// TIA Portal V18 export
VAR_GLOBAL   // PLC tag table "Default tag table"
   "Alarm Drive1" AT %I0.0 : Bool;
   "Alarm Drive 2" AT %I0.1 : Bool;
   setFlowRate AT %IW64 : Int;
   "AI on board(1)" AT %IW102 : Int;
   "preliminary empty signal component B1" AT %I0.6 : Bool;
   "Metering Start Foot Switch" AT %I1.2 : Bool;
   "Metering Start" AT %I1.3 : Bool;
   "Metering Stop" AT %I1.4 : Bool;
   "Metering Function Selection" AT %I2.0 : Bool;
   "Prerun Function" AT %I2.1 : Bool;
   "level empty signal component B1" AT %I0.7 : Bool;
   Flush AT %I2.2 : Bool;
   "Pressure sensor Pump Inlet A" AT %IW112 : Int;
   "Pressure Sensor Pump Inlet B" AT %IW114 : Int;
   "Pressure Sensor Pump Outlet A" AT %IW116 : Int;
   "Pressure Sensor Pump Outlet B" AT %IW118 : Int;
   "RPM PUMP A" AT %ID1008 : DInt;
   "RPM PUMP B" AT %ID1012 : DInt;
   "Level empty Signal component A1" AT %I0.3 : Bool;
   "program selection bit 3" AT %I2.6 : Bool;
   "preliminary empty signal component A1" AT %I0.2 : Bool;
   "Program selection bit0" AT %I2.3 : Bool;   //    {ExternalWritable false}
   "program selection bit 1" AT %I2.4 : Bool;
   "program selection bit2" AT %I2.5 : Bool;
   "Regenration Position Reached" AT %I1.5 : Bool;
   "reset pb" AT %I2.7 : Bool;
   "preliminary empty signal component A2" AT %I0.4 : Bool;
   "Level empty Signal component A2" AT %I0.5 : Bool;
   "preliminary empty signal component B2" AT %I1.0 : Bool;
   "level empty signal component B2" AT %I1.1 : Bool;
   "Level Sensor A" AT %IW120 : Int;
   "Level Sensor B" AT %IW122 : Int;
   "Pressure sensor Pump Inlet A_mA" AT %IW124 : Int;
   "Pressure Sensor Pump Inlet B_mA" AT %IW126 : Int;
   "emergency stop" AT %M3.5 : Bool;
   heater1 AT %IW144 : Int;
   heater2 AT %IW146 : Int;
   heater3 AT %IW148 : Int;
   heater4 AT %IW150 : Int;
   "Control ON" AT %I3.0 : Bool;
   "Control ON Led" AT %Q1.0 : Bool;
   "Reserve out3" AT %Q1.1 : Bool;
   "Metering Running" AT %Q2.2 : Bool;
   "ready to meter" AT %Q2.0 : Bool;
   "Metering Fault" AT %Q2.5 : Bool;
   "General Alarm" AT %Q2.1 : Bool;
   "Waiting for pre run" AT %Q2.3 : Bool;
   "metering Completed" AT %Q2.4 : Bool;
   "tower lamp yellow" AT %Q0.5 : Bool;
   "Reserve out0" AT %Q0.6 : Bool;
   "Reserve out1" AT %Q0.7 : Bool;
   "potlife error" AT %Q2.6 : Bool;
   "Reserve Output6" AT %Q2.7 : Bool;
   buzzer AT %Q0.4 : Bool;
   "Gear Pump A On_FWD" AT %Q0.0 : Bool;
   "Gear Pump B On_FWD" AT %Q0.2 : Bool;
   speedReference_ComponentB AT %QW130 : Int;
   speedReference_ComponentA AT %QW128 : Int;
   rampReference_ComponentA AT %QW132 : Int;
   rampReference_ComponentB AT %QW134 : Int;
   "Gear Pump A On_REW" AT %Q0.1 : Bool;
   "Gear Pump B On_REW" AT %Q0.3 : Bool;
   "Material 1 Temperature output" AT %Q3.0 : Bool;
   "Material 2 Temperature output" AT %Q3.1 : Bool;
   "Material 3 Temperature output" AT %Q3.2 : Bool;
   "Material 4 Temperature output" AT %Q3.3 : Bool;
   "gear Pump A fault" AT %M100.1 : Bool;
   "gear Pump B fault" AT %M100.2 : Bool;
   "Outlet Component A On" AT %M261.4 : Bool;
   "Outlet Component B On" AT %M200.4 : Bool;
   "program selection bit4" AT %M100.5 : Bool;
   "Agitator B Fault" AT %M100.3 : Bool;
   "Phase sequence relay Failure" AT %M100.4 : Bool;
   "Part Present sensor" AT %M100.0 : Bool;
   "Metering Ready" AT %M201.2 : Bool;
   "Tank A1 pressure" AT %MW240 : Int;
   "Tank A2 pressure" AT %MW242 : Int;
   "Tank B1 pressure" AT %MW244 : Int;
   "Tank Level A2" AT %MW248 : Int;
   "Gear Pump A Speed" AT %MW128 : Int;
   "Gear Pump B Speed" AT %MW130 : Int;
   "Mixer Speed" AT %MW208 : Int;
   "reserve  Analog output_0" AT %MW210 : Int;
   System_Byte AT %MB1 : Byte;
   FirstScan AT %M1.0 : Bool;
   DiagStatusUpdate AT %M1.1 : Bool;
   AlwaysTRUE AT %M1.2 : Bool;
   AlwaysFALSE AT %M1.3 : Bool;
   Clock_Byte AT %MB0 : Byte;
   Clock_10Hz AT %M0.0 : Bool;
   Clock_5Hz AT %M0.1 : Bool;
   "Clock_2.5Hz" AT %M0.2 : Bool;
   Clock_2Hz AT %M0.3 : Bool;
   "Clock_1.25Hz" AT %M0.4 : Bool;
   Clock_1Hz AT %M0.5 : Bool;
   "Clock_0.625Hz" AT %M0.6 : Bool;
   "Clock_0.5Hz" AT %M0.7 : Bool;
   "Fault register 1" AT %MW60 : Word;
   "Fault register 2" AT %MW62 : Word;
   "Fault register 3" AT %MW64 : Word;
   "Fault register 4" AT %MW66 : Word;
   "Fault register 5" AT %MW68 : Word;
   "A1-emergency stop active" AT %M61.0 : Bool;
   "A2-Pump A Drive Fault" AT %M61.1 : Bool;
   "A3-pump B drive Fault" AT %M61.2 : Bool;
   "A4-Agitator A1 fault" AT %M61.3 : Bool;
   "A5-Agitator A2 fault" AT %M61.4 : Bool;
   "A6-Tank A level sensor fault" AT %M61.5 : Bool;
   "A7-Tank B level sensor fault" AT %M61.6 : Bool;
   "A8-Pump A pressure sensor fault" AT %M61.7 : Bool;
   "A9-Pump B pressure sensor fault" AT %M60.0 : Bool;
   "A10-Tank A1 level sensor fault" AT %M60.1 : Bool;
   "A11-Tank A Filling Error" AT %M60.2 : Bool;
   "A12-Heater1 sensor fault" AT %M60.3 : Bool;
   "A13-Heater2 sensor fault" AT %M60.4 : Bool;
   "A14-Heater3 sensor fault" AT %M60.5 : Bool;
   "A15-Heater4 sensor fault" AT %M60.6 : Bool;
   "A16-Vaccum pump A fault" AT %M60.7 : Bool;
   "A17-Heater1 undertemperature" AT %M63.0 : Bool;
   "A18-Heater2 undertemperature" AT %M63.1 : Bool;
   "A19-Heater3 undertemperature" AT %M63.2 : Bool;
   "A20-Heater4 undertemperature" AT %M63.3 : Bool;
   "A21- Heater1 overtemperature" AT %M63.4 : Bool;
   "A22- Heater2 overtemperature" AT %M63.5 : Bool;
   "A23- Heater3 overtemperature" AT %M63.6 : Bool;
   "A24- Heater4 overtemperature" AT %M63.7 : Bool;
   "A25- Heater 8 pt100 discooneted" AT %M62.0 : Bool;
   "A26- Heater 9 pt100 discooneted" AT %M62.1 : Bool;
   "A27- Heater 10 pt100 discooneted" AT %M62.2 : Bool;
   "A28- Pump A over pressure" AT %M62.3 : Bool;
   "A29-pump B Over pressure" AT %M62.4 : Bool;
   "A30-Tank A1 Level Empty" AT %M62.5 : Bool;
   "A31-Tank A2 Level Empty" AT %M62.6 : Bool;
   "A32-Tank B Level Empty" AT %M62.7 : Bool;
   "A33-Tank A1 low level" AT %M65.0 : Bool;
   "A34-Tank A2 low level" AT %M65.1 : Bool;
   "A35-Tank B low level" AT %M65.2 : Bool;
   "A36-Pump A lower pressure" AT %M65.3 : Bool;
   "A37-Pump B lower pressure" AT %M65.4 : Bool;
   "A38-A material Supply fault" AT %M65.5 : Bool;
   "A39-B material Supply fault" AT %M65.6 : Bool;
   "A40-Potlife elapsed Change static mixer" AT %M65.7 : Bool;
   "A41- Heater 1 temperature Low" AT %M64.0 : Bool;
   "A42- Heater 2 temperature Low" AT %M64.1 : Bool;
   "A43- Heater 3 temperature Low" AT %M64.2 : Bool;
   "A44- Heater 4 temperature Low" AT %M64.3 : Bool;
   "A45- Heater 5 temperature Low" AT %M64.4 : Bool;
   "A46- Heater 6 temperature Low" AT %M64.5 : Bool;
   "A47- Heater 7 temperature Low" AT %M64.6 : Bool;
   "A48- Heater 8 temperature Low" AT %M64.7 : Bool;
   "A49- heater 9 temperature low" AT %M67.0 : Bool;
   "A50- heater 10 temperature low" AT %M67.1 : Bool;
   "A51- heater 1 temperature high" AT %M67.2 : Bool;
   "A52- heater 2 temperature high" AT %M67.3 : Bool;
   "A53- heater 3 temperature high" AT %M67.4 : Bool;
   "A54- heater 4 temperature high" AT %M67.5 : Bool;
   "A55- heater 5 temperature high" AT %M67.6 : Bool;
   "A56- heater 6 temperature high" AT %M67.7 : Bool;
   "A57- heater  7 temperature high" AT %M66.0 : Bool;
   "A58- heater 8 temperature high" AT %M66.1 : Bool;
   "A59- heater 9 temperature high" AT %M66.2 : Bool;
   "A60- heater 10 temperature high" AT %M66.3 : Bool;
   "A61- refilling failed Tank A1" AT %M66.4 : Bool;
   "A62-Error flowrate" AT %M66.5 : Bool;
   "A63- refilling failed Tank B" AT %M66.6 : Bool;
   Ack_A1 AT %M341.0 : Bool;
   Ack_A2 AT %M341.1 : Bool;
   Ack_A3 AT %M341.2 : Bool;
   Ack_A4 AT %M341.3 : Bool;
   Ack_A5 AT %M341.4 : Bool;
   Ack_A6 AT %M341.5 : Bool;
   Ack_A7 AT %M341.6 : Bool;
   Ack_A8 AT %M341.7 : Bool;
   Ack_A9 AT %M342.0 : Bool;
   Ack_A10 AT %M342.1 : Bool;
   Ack_A11 AT %M342.2 : Bool;
   Ack_A12 AT %M342.3 : Bool;
   Ack_A13 AT %M342.4 : Bool;
   Ack_A14 AT %M342.5 : Bool;
   Ack_A15 AT %M342.6 : Bool;
   Ack_A16 AT %M342.7 : Bool;
   Ack_A17 AT %M343.0 : Bool;
   Ack_A18 AT %M343.1 : Bool;
   Ack_A19 AT %M343.2 : Bool;
   Ack_A20 AT %M343.3 : Bool;
   Ack_A21 AT %M343.4 : Bool;
   Ack_A22 AT %M343.5 : Bool;
   Ack_A23 AT %M343.6 : Bool;
   Ack_A24 AT %M343.7 : Bool;
   Ack_A25 AT %M344.0 : Bool;
   Ack_A26 AT %M344.1 : Bool;
   Ack_A27 AT %M344.2 : Bool;
   Ack_A28 AT %M344.3 : Bool;
   Ack_A29 AT %M344.4 : Bool;
   Ack_A30 AT %M344.5 : Bool;
   Ack_A31 AT %M344.6 : Bool;
   Ack_A32 AT %M344.7 : Bool;
   Ack_A33 AT %M345.0 : Bool;
   Ack_A34 AT %M345.1 : Bool;
   Ack_A35 AT %M345.2 : Bool;
   Ack_A36 AT %M345.3 : Bool;
   Ack_A37 AT %M345.4 : Bool;
   Ack_A38 AT %M345.5 : Bool;
   Ack_A39 AT %M345.6 : Bool;
   Ack_A40 AT %M345.7 : Bool;
   Ack_A41 AT %M346.0 : Bool;
   Ack_A42 AT %M346.1 : Bool;
   Ack_A43 AT %M346.2 : Bool;
   Ack_A44 AT %M346.3 : Bool;
   Ack_A45 AT %M346.4 : Bool;
   Ack_A46 AT %M346.5 : Bool;
   Ack_A47 AT %M346.6 : Bool;
   Ack_A48 AT %M346.7 : Bool;
   Ack_A49 AT %M347.0 : Bool;
   Ack_A50 AT %M347.1 : Bool;
   Ack_A51 AT %M347.2 : Bool;
   Ack_A52 AT %M347.3 : Bool;
   Ack_A53 AT %M347.4 : Bool;
   Ack_A54 AT %M347.5 : Bool;
   Ack_A55 AT %M347.6 : Bool;
   Ack_A56 AT %M347.7 : Bool;
   Ack_A57 AT %M348.0 : Bool;
   Ack_A58 AT %M348.1 : Bool;
   Ack_A59 AT %M348.2 : Bool;
   Ack_A60 AT %M348.3 : Bool;
   Ack_A61 AT %M348.4 : Bool;
   Ack_A62 AT %M348.5 : Bool;
   Ack_A63 AT %M348.6 : Bool;
   Ack_A64 AT %M348.7 : Bool;
   Ack_A65 AT %M349.0 : Bool;
   Ack_A66 AT %M349.1 : Bool;
   Ack_A67 AT %M349.2 : Bool;
   Ack_A68 AT %M349.3 : Bool;
   Ack_A69 AT %M349.4 : Bool;
   Ack_hmi AT %M39.0 : Bool;
   Ack_site AT %M39.1 : Bool;
   Ack_PB AT %M39.2 : Bool;
   Fault_Ack_ONS AT %M39.3 : Bool;
   Tag_1 AT %M21.0 : Bool;
   Tag_2 AT %M4.1 : Bool;
   Ack_hmi_ons AT %M39.4 : Bool;
   "1sec_pulse" AT %M2.0 : Bool;
   "transperant backround" AT %M5.0 : Bool;
   "error count" AT %MD6 : UDInt;
   "A66-Tank A1 over pressure" AT %M69.1 : Bool;
   "A67-Tank A2 over pressure" AT %M69.2 : Bool;
   "A68-Tank B1 over pressure" AT %M69.3 : Bool;
   "Pgm No site" AT %MW23 : Int;
   "Pgm selection Bit memory 1" AT %M23.0 : Bool;
   "Pgm selection Bit memory 2" AT %M23.1 : Bool;
   "Pgm selection Bit memory 3" AT %M23.2 : Bool;
   "Pgm selection Bit memory 4" AT %M23.4 : Bool;
   "A69-mixer element break" AT %M69.4 : Bool;
   "Tank B2 pressure" AT %MW246 : Int;
   "Tank Level B2" AT %MW250 : Int;
   "VC1 new Pulse" AT %MD500 : DWord;
   "VC1 OLD Pulse" AT %MD504 : DWord;
   "VC2 new Pulse" AT %MD508 : DWord;
   "VC2 OLD Pulse" AT %MD512 : DWord;
   "VC1 Frequency" AT %MD516 : Real;
   "VC2 Frequency" AT %MD520 : Real;
   "VC1 Pulse in 1HZ" AT %MD524 : Real;
   "VC2 Pulse in 1HZ" AT %MD528 : Real;
   Tag_3 AT %MD1000 : DInt;
   Ack_A70 AT %M349.5 : Bool;
   Ack_A71 AT %M349.6 : Bool;
   Ack_A72 AT %M349.7 : Bool;
   Ack_A73 AT %M350.0 : Bool;
   "A70-mixing ratio low  warning" AT %M69.5 : Bool;
   "A71-mixing ratio high warning" AT %M69.6 : Bool;
   "A72-mixing ratio low fault" AT %M69.7 : Bool;
   "A89-Level Empty Drum B2" AT %M70.0 : Bool;
   "ready to power on servo" AT %M2.1 : Bool;
   "Pump Ready A1" AT %M100.6 : Bool;
   "Pump Ready A2" AT %M100.7 : Bool;
   "Pump Ready B1" AT %M101.0 : Bool;
   "Pump Ready B2" AT %M101.1 : Bool;
   Ack_A74 AT %M350.1 : Bool;
   Ack_A75 AT %M350.2 : Bool;
   Ack_A76 AT %M350.3 : Bool;
   Ack_A77 AT %M350.4 : Bool;
   Ack_A78 AT %M350.5 : Bool;
   Ack_A79 AT %M350.6 : Bool;
   Ack_A80 AT %M350.7 : Bool;
   Ack_A81 AT %M351.0 : Bool;
   Ack_A82 AT %M351.1 : Bool;
   Ack_A83 AT %M351.2 : Bool;
   Ack_A84 AT %M351.3 : Bool;
   Ack_A85 AT %M351.4 : Bool;
   Ack_A86 AT %M351.5 : Bool;
   Ack_A87 AT %M351.6 : Bool;
   Ack_A88 AT %M351.7 : Bool;
   Ack_A89 AT %M352.0 : Bool;
   Ack_A90 AT %M352.1 : Bool;
   Ack_A91 AT %M352.2 : Bool;
   Ack_A92 AT %M352.3 : Bool;
   Ack_A93 AT %M352.4 : Bool;
   Ack_A94 AT %M352.5 : Bool;
   Ack_A95 AT %M352.6 : Bool;
   Ack_A96 AT %M352.7 : Bool;
   Ack_A97 AT %M353.0 : Bool;
   Ack_A98 AT %M353.1 : Bool;
   Ack_A99 AT %M353.2 : Bool;
   Ack_A100 AT %M353.3 : Bool;
   Ack_A101 AT %M353.4 : Bool;
   Ack_A102 AT %M353.5 : Bool;
   Ack_A103 AT %M353.6 : Bool;
   Ack_A104 AT %M353.7 : Bool;
   Ack_A105 AT %M354.0 : Bool;
   Ack_A106 AT %M354.1 : Bool;
   Ack_A107 AT %M354.2 : Bool;
   Ack_A108 AT %M354.3 : Bool;
   Ack_A109 AT %M354.4 : Bool;
   Ack_A110 AT %M354.5 : Bool;
   Ack_A111 AT %M354.6 : Bool;
   Ack_A112 AT %M355.0 : Bool;
   Ack_A113 AT %M355.1 : Bool;
   Ack_A114 AT %M355.2 : Bool;
   Ack_A115 AT %M355.3 : Bool;
   Ack_A116 AT %M355.4 : Bool;
   Ack_A117 AT %M355.5 : Bool;
   Ack_A118 AT %M355.6 : Bool;
   Ack_A119 AT %M355.7 : Bool;
   Ack_A120 AT %M356.0 : Bool;
   Ack_A121 AT %M356.1 : Bool;
   Ack_A122 AT %M356.2 : Bool;
   Ack_A123 AT %M356.3 : Bool;
   Ack_A124 AT %M356.4 : Bool;
   Ack_A125 AT %M356.5 : Bool;
   Ack_A126 AT %M356.6 : Bool;
   Ack_A127 AT %M356.7 : Bool;
   Ack_A128 AT %M357.0 : Bool;
   Ack_A129 AT %M357.1 : Bool;
   Ack_A130 AT %M357.2 : Bool;
   Ack_A131 AT %M357.3 : Bool;
   Ack_A132 AT %M357.4 : Bool;
   Ack_A133 AT %M357.5 : Bool;
   Ack_A134 AT %M357.6 : Bool;
   Ack_A135 AT %M357.7 : Bool;
   Ack_A136 AT %M358.0 : Bool;
   Ack_A137 AT %M358.1 : Bool;
   Ack_A138 AT %M358.2 : Bool;
   Ack_A139 AT %M358.3 : Bool;
   Ack_A140 AT %M358.4 : Bool;
   Ack_A141 AT %M358.5 : Bool;
   Ack_A142 AT %M358.6 : Bool;
   Ack_A143 AT %M358.7 : Bool;
   "Fault register 6" AT %MW70 : Word;
   "Fault register 7" AT %MW72 : Word;
   "Fault register 8" AT %MW74 : Word;
   "Fault register 9" AT %MW76 : Word;
   Ack_A144 AT %M359.0 : Bool;
   Ack_A145 AT %M359.1 : Bool;
   Ack_A146 AT %M359.2 : Bool;
   Ack_A147 AT %M359.3 : Bool;
   Ack_A148 AT %M359.4 : Bool;
   Ack_A149 AT %M359.5 : Bool;
   Ack_A150 AT %M359.6 : Bool;
   Ack_A151 AT %M359.7 : Bool;
   Ack_A152 AT %M360.0 : Bool;
   Ack_A154 AT %M360.2 : Bool;
   Ack_A155 AT %M360.3 : Bool;
   Ack_A156 AT %M360.4 : Bool;
   Ack_A157 AT %M360.5 : Bool;
   Ack_A158 AT %M360.6 : Bool;
   Ack_A159 AT %M360.7 : Bool;
   Ack_A160 AT %M361.0 : Bool;
   "A82-Level Low Drum A1" AT %M71.1 : Bool;
   "A83-Level Low Drum B1" AT %M71.2 : Bool;
   "A84-Level Low Drum A2" AT %M71.3 : Bool;
   "A85-Level Low Drum B2" AT %M71.4 : Bool;
   "A86-Level Empty Drum A1" AT %M71.5 : Bool;
   "A87-Level Empty Drum B1" AT %M71.6 : Bool;
   "A88-Level Empty Drum A2" AT %M71.7 : Bool;
   Ack_A168 AT %M361.1 : Bool;
   Ack_A169 AT %M361.2 : Bool;
   Ack_A170 AT %M361.3 : Bool;
   Ack_A171 AT %M361.4 : Bool;
   Ack_A172 AT %M361.5 : Bool;
   Ack_A173 AT %M361.6 : Bool;
   Ack_A174 AT %M361.7 : Bool;
   Ack_A175 AT %M362.0 : Bool;
   Ack_A176 AT %M362.1 : Bool;
   Ack_A177 AT %M362.2 : Bool;
   Ack_A178 AT %M362.3 : Bool;
   Ack_A179 AT %M362.4 : Bool;
   Ack_A180 AT %M362.5 : Bool;
   Ack_A181 AT %M362.6 : Bool;
   Ack_A182 AT %M362.7 : Bool;
   Ack_A183 AT %M363.0 : Bool;
   Ack_A184 AT %M363.1 : Bool;
   Ack_A185 AT %M363.2 : Bool;
   Ack_A186 AT %M363.3 : Bool;
   Ack_A187 AT %M363.4 : Bool;
   Ack_A188 AT %M363.5 : Bool;
   "Fault register 10" AT %MW32 : Word;
   "A74-Level Low Pressure Vessel A" AT %M68.1 : Bool;
   "A75-Level Low Pressure Vessel B" AT %M68.2 : Bool;
   "A76-Level Empty Pressure Vessel A" AT %M68.3 : Bool;
   "A77-Level Empty Pressure Vessel B" AT %M68.4 : Bool;
   "A78-Level Low Catridge A" AT %M68.5 : Bool;
   "A79-Level Low Catridge B" AT %M68.6 : Bool;
   "A80-Level Empty Catridge A" AT %M68.7 : Bool;
   Tag_4 AT %M73.0 : Bool;
   Tag_5 AT %M73.1 : Bool;
   Tag_6 AT %M73.2 : Bool;
   Tag_7 AT %M73.3 : Bool;
   Tag_8 AT %M73.4 : Bool;
   Tag_9 AT %M73.5 : Bool;
   Tag_10 AT %M73.6 : Bool;
   Tag_11 AT %M73.7 : Bool;
   "A90 Pressure sensor Pump A Outlet Fault" AT %M72.0 : Bool;
   "A91 Pressure sensor Pump B Outlet Fault" AT %M72.1 : Bool;
   "A92 Over pressure A outlet" AT %M72.2 : Bool;
   "A93 Over pressure B outlet" AT %M72.3 : Bool;
   "A94- Pump A Outlet Under Pressure" AT %M72.4 : Bool;
   "A95- Pump B Outlet Under Pressure" AT %M72.5 : Bool;
   Tag_18 AT %M72.6 : Bool;
   Tag_19 AT %M72.7 : Bool;
   Tag_20 AT %M75.0 : Bool;
   Tag_21 AT %M75.1 : Bool;
   Tag_22 AT %M75.2 : Bool;
   Tag_23 AT %M75.3 : Bool;
   Tag_24 AT %M75.4 : Bool;
   Tag_25 AT %M75.5 : Bool;
   Tag_26 AT %M75.6 : Bool;
   Tag_27 AT %M75.7 : Bool;
   Tag_28 AT %M74.0 : Bool;
   Tag_29 AT %M74.1 : Bool;
   Tag_30 AT %M74.2 : Bool;
   Tag_31 AT %M74.3 : Bool;
   Tag_32 AT %M74.4 : Bool;
   Tag_33 AT %M74.5 : Bool;
   Tag_34 AT %M74.6 : Bool;
   Tag_35 AT %M74.7 : Bool;
   Tag_36 AT %M77.0 : Bool;
   Tag_37 AT %M77.1 : Bool;
   Tag_38 AT %M77.2 : Bool;
   Tag_39 AT %M77.3 : Bool;
   Tag_40 AT %M77.4 : Bool;
   Tag_41 AT %M77.5 : Bool;
   Tag_42 AT %M77.6 : Bool;
   Tag_43 AT %M77.7 : Bool;
   Tag_44 AT %M76.0 : Bool;
   Tag_45 AT %M76.1 : Bool;
   Tag_46 AT %M76.2 : Bool;
   Tag_47 AT %M76.3 : Bool;
   Tag_48 AT %M76.4 : Bool;
   Tag_49 AT %M76.5 : Bool;
   Tag_50 AT %M76.6 : Bool;
   Tag_51 AT %M76.7 : Bool;
   Ack_A153 AT %M360.1 : Bool;
   "Inlet Component A On" AT %M261.2 : Bool;
   "Inlet Component B On" AT %M261.3 : Bool;
   "Agitator B" AT %M200.3 : Bool;
   "Material refilling A" AT %M200.5 : Bool;
   "Material refilling B" AT %M200.6 : Bool;
   "Refilling Pump A" AT %M200.7 : Bool;
   "Refilling Pump B" AT %M201.0 : Bool;
   "Reserve Output 3" AT %M201.1 : Bool;
   "Pressure Release A" AT %M200.2 : Bool;
   "Pressure Release B" AT %M201.3 : Bool;
   "A64- No siganl RPM sensor A" AT %M70.2 : Bool;
   "A65- No siganl RPM sensor B" AT %M70.3 : Bool;
   "A70-Warning mixing ratio low" AT %M70.4 : Bool;
   "A71- warning Mixing Ratio high" AT %M70.5 : Bool;
   "A72- Error Mixing ratio Low" AT %M70.6 : Bool;
   "A73- Error Mixing Ratio high" AT %M70.7 : Bool;
   Tag_52 AT %M30.0 : Bool;
   Tag_53 AT %M30.1 : Bool;
   Tag_54 AT %M500.0 : Bool;
   tnp AT %M2.2 : Bool;
   "PID A setpoint scaled" AT %MD10 : Real;
   "PID A input scaled" AT %MD14 : Real;
   "PID B setpoint scaled" AT %MD34 : Real;
   "PID B input scaled" AT %MD40 : Real;
   dummy1 AT %M2.3 : Bool;
   "RTD OUTPUT" AT %MD44 : Real;
   "RTD OUTPUT1" AT %MD48 : Real;
   "prg no sel" AT %MW18 : Int;
   "SD Logg" AT %MD52 : UDInt;
   "SD LOG TRIGGER" AT %M2.5 : Bool;
   "USB Logg" AT %MD140 : UDInt;
   "USB LOG TRIGGER" AT %M2.6 : Bool;
   "A81-Level Empty Catridge B" AT %M71.0 : Bool;
   TempPE1 AT %M2.7 : Bool;
   TempPE2 AT %M3.0 : Bool;
   temps AT %MD102 : Real;
   temp_unitsel AT %MW56 : Int;
   test AT %M3.1 : Bool;
   snuffback_completed AT %M3.2 : Bool;
   temp_dispese_qty AT %MD26 : Real;
   RatioCheck_status AT %MW78 : Int;
   actual_gramA_Old AT %MD106 : Real;
   actual_gramB_Old AT %MD110 : Real;
   Function_snuffback_selected AT %M3.3 : Bool;
   start_snuffback AT %M3.4 : Bool;
   "Fault display register 1" AT %MW80 : Word;
   "Fault display register 2" AT %MW82 : Word;
   "Fault display register 3" AT %MW84 : Word;
   "Fault display register 4" AT %MW86 : Word;
   "Fault display register 5" AT %MW88 : Word;
   "Fault display register 6" AT %MW90 : Word;
   "Fault display register 7" AT %MW92 : Word;
   machine_on AT %M2.4 : Bool;
   estop AT %I3.1 : Bool;
END_VAR
